// TwinCAT 3 PLC project PLC1
// ProgramVersion: 3.1.4023.0
// libraries:
//   Tc2_Standard, * (Beckhoff Automation GmbH)
//   Tc2_System, * (Beckhoff Automation GmbH)
//   Tc3_Module, * (Beckhoff Automation GmbH)
// project tree:
//   / PlcTask.TcTTO
//   POUs/ MAIN.TcPOU
// real-time tasks:
//   TASK PlcTask: cycle T#10ms, priority 6, ADS port 350

CONFIGURATION PLC1
    RESOURCE PLC ON TwinCAT3
        TASK PlcTask(INTERVAL := T#10ms, PRIORITY := 6);
        PROGRAM MAIN WITH PlcTask : MAIN;
    END_RESOURCE
END_CONFIGURATION

// ---- POUs/MAIN.TcPOU
PROGRAM MAIN
VAR
	xStart : BOOL := FALSE;
	xEStop : BOOL := FALSE; 
	xMotor : BOOL := FALSE;
	xEnable : BOOL := FALSE;
	XLocked : BOOL := FALSE;
	xInTimer : BOOL:= FALSE;
	fbTMR : TON;
END_VAR



xEnable := (xStart OR xEnable) AND NOT xEStop AND NOT xLocked;


IF xEStop THEN 
	
	xLocked := TRUE;
	xInTimer := TRUE;
	
END_IF

fbTMR(IN := xInTimer,
	PT := T#10S );
	

IF fbTMR.Q THEN
	
	xLocked := FALSE;
	xInTimer := FALSE;

END_IF

END_PROGRAM
